VAR_GLOBAL
END_VAR

(* stored: Version 1.1.0.1, ProductVersion 3.1.4022.12
   GVL GVL_VARIABLES: Id {89f0e23b-0303-4f40-ba76-e23c3ad240c9} *)
